// Gets the upper bound index of the array of specified type.
FUNCTION F_GetDIntArrayUpperBound : T_Position // The upper bound index of the specified array.
VAR_IN_OUT
	arArray : ARRAY[*] OF DINT; // The array to query.
END_VAR

F_GetDIntArrayUpperBound := UPPER_BOUND(arArray, 1);

END_FUNCTION

(* stored: Version 1.1.0.1
   POU F_GetDIntArrayUpperBound: Id {cadc1d9e-cd55-0359-3b20-515458cb188e}, SpecialFunc None *)
